PROGRAM PRG_Controller_TEST
VAR
END_VAR

END_PROGRAM

(* stored: Version 1.1.0.1, ProductVersion 3.1.4024.13
   POU PRG_Controller_TEST: Id {fa9678cb-1344-4880-8f88-578d5e8978bd}, SpecialFunc None *)
